{attribute 'qualified_only'}
VAR_GLOBAL
	
END_VAR

(* stored: Version 1.1.0.1
   GVL IO_VFDs: Id {9aff624f-d785-43b7-bbb2-8323195aaf84} *)
